SUBAPPLICATION ACTION_SERVER_STATUS
  (* Standard: 61499-2 *)
  (* Version 1.0, 2023-04-02, Tim Hesse *)
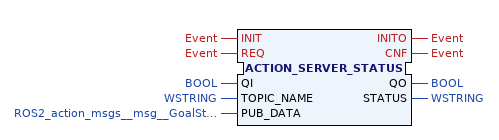
  EVENT_INPUT
    INIT; (* Initialization Request *)
    REQ;
  END_EVENT
  EVENT_OUTPUT
    INITO; (* Initialization Confirm *)
    CNF;
  END_EVENT
  VAR_INPUT
    QI : BOOL; (* Input event qualifier *)
    TOPIC_NAME : WSTRING;
    PUB_DATA : ROS2_action_msgs__msg__GoalStatusArray;
  END_VAR
  VAR_OUTPUT
    QO : BOOL; (* Output event qualifier *)
    STATUS : WSTRING;
  END_VAR
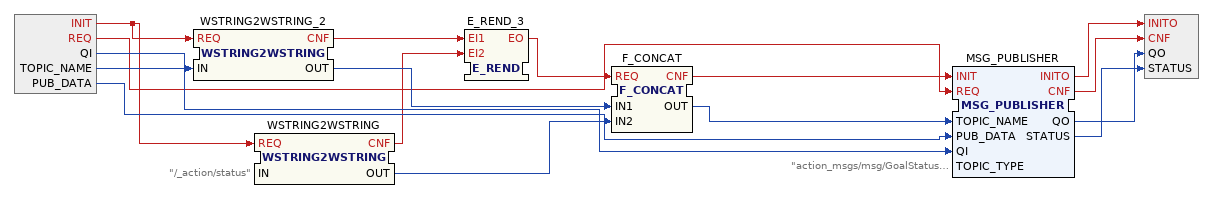
  FBS
    WSTRING2WSTRING_2 : WSTRING2WSTRING;
    F_CONCAT : F_CONCAT;
    E_REND_3 : E_REND;
    WSTRING2WSTRING : WSTRING2WSTRING(IN := "/_action/status");
  END_FBS
  SUBAPPS
    MSG_PUBLISHER : MSG_PUBLISHER(TOPIC_TYPE := "action_msgs/msg/GoalStatusArray");
  END_SUBAPPS
  EVENT_CONNECTIONS
    E_REND_3.EO TO F_CONCAT.REQ;
    WSTRING2WSTRING_2.CNF TO E_REND_3.EI1;
    WSTRING2WSTRING.CNF TO E_REND_3.EI2;
    INIT TO WSTRING2WSTRING_2.REQ;
    INIT TO WSTRING2WSTRING.REQ;
    F_CONCAT.CNF TO MSG_PUBLISHER.INIT;
    REQ TO MSG_PUBLISHER.REQ;
    MSG_PUBLISHER.INITO TO INITO;
    MSG_PUBLISHER.CNF TO CNF;
  END_CONNECTIONS
  DATA_CONNECTIONS
    WSTRING2WSTRING_2.OUT TO F_CONCAT.IN1;
    WSTRING2WSTRING.OUT TO F_CONCAT.IN2;
    F_CONCAT.OUT TO MSG_PUBLISHER.TOPIC_NAME;
    TOPIC_NAME TO WSTRING2WSTRING_2.IN;
    PUB_DATA TO MSG_PUBLISHER.PUB_DATA;
    QI TO MSG_PUBLISHER.QI;
    MSG_PUBLISHER.QO TO QO;
    MSG_PUBLISHER.STATUS TO STATUS;
  END_CONNECTIONS
END_SUBAPPLICATION
